INTERFACE I_Mfr_Event

METHOD Acknowledge
END_METHOD

PROPERTY Active : BOOL
GET
END_GET
END_PROPERTY

PROPERTY Message : T_MaxString
GET
END_GET
END_PROPERTY

{attribute 'hide'}
PROPERTY Next : I_Mfr_Event
GET
END_GET
SET
END_SET
END_PROPERTY

PROPERTY Severity : E_Mfr_NotifySeverity
GET
END_GET
END_PROPERTY

PROPERTY Title : STRING
GET
END_GET
END_PROPERTY

END_INTERFACE

(* stored: Version 1.1.0.1
   Itf I_Mfr_Event: Id {d8d3a27e-3fb4-4fd1-9174-dc0d7cf4b95d}
   Folder [Internal]: Id {ba28ae2e-6e81-4932-8ef9-1640e1b0d1b8}
   Method Acknowledge: Id {d19a932b-47de-4942-8ec4-bc38f6d0d62f}
   Property Active: Id {7d739ef1-4f96-4039-af4f-bd758d8effa4}
   Get Get: Id {10e6464d-881f-42ec-a2bf-d3eca325c573}
   Property Message: Id {9a84164a-0c8e-4f95-acea-0d1dec31bbb6}
   Get Get: Id {7c19bae1-e887-40b5-9065-c216763186c1}
   Property Next: Id {ee64735e-bdf3-42ca-b21d-e8683385bc6f}
   Get Get: Id {a32292f4-48de-4671-9847-49e81cdfdcf1}
   Set Set: Id {c2fbb5a3-b5d8-4e08-aa24-dc1ecfdc75a8}
   Property Severity: Id {d6a17e07-3e60-4887-bf90-510e063c403f}
   Get Get: Id {95aff632-5681-4f87-97ef-d5ece2c96aa3}
   Property Title: Id {2d395dc2-8f41-4f16-ae4c-6fe95a040920}
   Get Get: Id {fa5d78c5-77d8-44bc-93a6-6a49d0c6ba50} *)
